# EPICS StreamDevice protocol: TopConApp/Db/Regatron.proto
Terminator = CR;

#  // [IGBT,Rectfier,PCB]
#  getTemperatures
#  // [Voltage,Current,Power,Res,State]
#  getModReadings
#  getSysReadings
#  // [..Error,..Warning] T_ErrorTree32
#  getModTree
#  getSysTree
#  // [..ErrorTree, ..WarnTree]\n
getArray{ separator=','; out "\$1"; in  "\$1 [%f]"; }

#  getModuleId
#  getModControlMode
#  getSysControlMode
#  getControlInput
#  getDCLinkVoltage
#  getPrimaryCurrent
getFloat{ out "\$1"; in  "\$1 %f"; }

#  getDSPVersion
#  getDLLVersion
#  getBootloaderVersion
#  getModulatorVersion
#  getPheripherieVersion
getString{ out "\$1"; in  "\$1 %s"; }

#  cmdStoreParam
#  cmdClearErrors
cmd{ out "\$1"; in  "\$1 ACK"; }
